// TwinCAT 3 PLC project PLCStudent
// ProgramVersion: 3.1.4022.3
// libraries:
//   Tc2_Standard, * (Beckhoff Automation GmbH)
//   Tc2_System, * (Beckhoff Automation GmbH)
//   Tc3_Module, * (Beckhoff Automation GmbH)
// project tree:
//   GVLs/ GVL.TcGVL
//   / PlcTask.TcTTO
//   POUs/ MAIN.TcPOU, PushPopFB.TcPOU, SFCMotor.TcPOU
// (motion and I/O tree: see PLC project plcsim)
// real-time tasks:
//   TASK PlcTask: cycle T#20ms, priority 20, ADS port 350
// variable links:
//   PLCSim/PLCSim Instance <-> PLCStudent/PLCStudent Instance
//     PlcTask Inputs/GVL.iiDisplayElevat <-> PlcTask Outputs/GVL.qiDispElevat
//     PlcTask Inputs/GVL.ixDoorClose <-> PlcTask Outputs/GVL.qxDoorClose
//     PlcTask Inputs/GVL.ixLampElevat1 <-> PlcTask Outputs/GVL.qxLampElevat1
//     PlcTask Inputs/GVL.ixLampElevat2 <-> PlcTask Outputs/GVL.qxLampElevat2
//     PlcTask Inputs/GVL.ixLampElevat3 <-> PlcTask Outputs/GVL.qxLampElevat3
//     PlcTask Inputs/GVL.ixLampLevel1 <-> PlcTask Outputs/GVL.qxLampLevel1
//     PlcTask Inputs/GVL.ixLampLevel2 <-> PlcTask Outputs/GVL.qxLampLevel2
//     PlcTask Inputs/GVL.ixLampLevel3 <-> PlcTask Outputs/GVL.qxLampLevel3
//     PlcTask Inputs/GVL.ixMotorDown <-> PlcTask Outputs/GVL.qxMotorDown
//     PlcTask Inputs/GVL.ixMotorUp <-> PlcTask Outputs/GVL.qxMotorUp
//     PlcTask Outputs/GVL.qxButtElevat1 <-> PlcTask Inputs/GVL.ixButtElevat1
//     PlcTask Outputs/GVL.qxButtElevat2 <-> PlcTask Inputs/GVL.ixButtElevat2
//     PlcTask Outputs/GVL.qxButtElevat3 <-> PlcTask Inputs/GVL.ixButtElevat3
//     PlcTask Outputs/GVL.qxButtGreen <-> PlcTask Inputs/GVL.ixButtGreen
//     PlcTask Outputs/GVL.qxButtLevel1 <-> PlcTask Inputs/GVL.ixButtLevel1
//     PlcTask Outputs/GVL.qxButtLevel2 <-> PlcTask Inputs/GVL.ixButtLevel2
//     PlcTask Outputs/GVL.qxButtLevel3 <-> PlcTask Inputs/GVL.ixButtLevel3
//     PlcTask Outputs/GVL.qxButtRed <-> PlcTask Inputs/GVL.ixButtRed
//     PlcTask Outputs/GVL.qxDoorClosed <-> PlcTask Inputs/GVL.ixDoorClosed
//     PlcTask Outputs/GVL.qxDoorOpen <-> PlcTask Inputs/GVL.ixDoorOpen
//     PlcTask Outputs/GVL.qxElevatLevel1 <-> PlcTask Inputs/GVL.ixElevatLevel1
//     PlcTask Outputs/GVL.qxElevatLevel2 <-> PlcTask Inputs/GVL.ixElevatLevel2
//     PlcTask Outputs/GVL.qxElevatLevel3 <-> PlcTask Inputs/GVL.ixElevatLevel3

CONFIGURATION PLCStudent
    RESOURCE PLC ON TwinCAT3
        TASK PlcTask(INTERVAL := T#20ms, PRIORITY := 20);
        PROGRAM MAIN WITH PlcTask : MAIN;
    END_RESOURCE
END_CONFIGURATION

// ---- GVLs/GVL.TcGVL
{attribute 'qualified_only'}
VAR_GLOBAL
//Input to PLC from process
	ixButtLevel1		AT %I*:	BOOL;		(* Button at level 1 *)
	ixButtLevel2		AT %I*:	BOOL;		(* Button at level 2 *)
	ixButtLevel3		AT %I*:	BOOL;		(* Button at level 3 *)

	ixButtElevat1		AT %I*:	BOOL;		(* Button 1 inside elevator *)
	ixButtElevat2		AT %I*:	BOOL;		(* Button 2 inside elevator *)
	ixButtElevat3		AT %I*:	BOOL;		(* Button 3 inside elevator *)

	ixButtGreen 		AT %I*:	BOOL;		(* Green button *)
	ixButtRed			AT %I*:	BOOL;		(* Red button, normally closed *)

	ixElevatLevel1 		AT %I*: BOOL;		(* Sensor at level 1 for elevator presence *)
	ixElevatLevel2 		AT %I*: BOOL;		(* Sensor at level 2 for elevator presence *)
	ixElevatLevel3 		AT %I*: BOOL;		(* Sensor at level 3 for elevator presence *)

	ixDoorClosed		AT %I*: BOOL;		(* Sensor for door closed *)
	ixDoorOpen			AT %I*:	BOOL;		(* Sensor for door open *)

//Output from PLC to process
	qxLampLevel1		AT %Q*:	BOOL;		(* Lamp at level 1*)
	qxLampLevel2		AT %Q*:	BOOL;		(* Lamp at level 2*)
	qxLampLevel3		AT %Q*:	BOOL;		(* Lamp at level 3*)

	qxLampElevat1 		AT %Q*:	BOOL;		(* Lamp 1 inside elevator *)
	qxLampElevat2 		AT %Q*:	BOOL;		(* Lamp 2 inside elevator *)
	qxLampElevat3 		AT %Q*:	BOOL;		(* Lamp 3 inside elevator *)

	qxMotorDown			AT %Q*:	BOOL;		(* Run motor down *)
	qxMotorUp			AT %Q*:	BOOL;		(* Run motor up *)

	qxDoorClose			AT %Q*:	BOOL;		(* Close door and keep it closed *)
	qiDispElevat 		AT %Q*:	UINT;		(* Integer display inside elevator *)
END_VAR

// ---- POUs/MAIN.TcPOU
PROGRAM MAIN
VAR
	
END_VAR

SFCMotor();

END_PROGRAM

// ---- POUs/SFCMotor.TcPOU
PROGRAM SFCMotor
VAR
	PushPopFB_0: PushPopFB;
	TargFloor: UINT;
	OutputFloor: UINT;
	MemoryMotor: UINT;

END_VAR
VAR // added by the converter: edge detectors and wires of the graphical bodies
    _rt1, _rt2, _rt3 : R_TRIG;
    _w1, _w2, _w3 : BOOL;
END_VAR

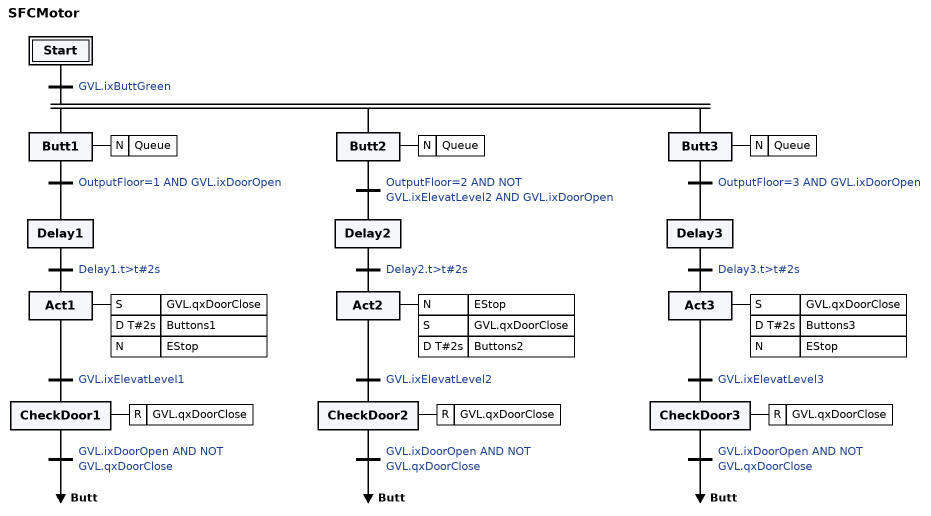
INITIAL_STEP Start:
END_STEP
TRANSITION FROM Start TO (Butt1, Butt2, Butt3)
    := GVL.ixButtGreen;
END_TRANSITION
STEP Butt1:
    Queue(N);
END_STEP
STEP Butt2:
    Queue(N);
END_STEP
TRANSITION FROM Butt2 TO Delay2
    := OutputFloor=2 AND NOT GVL.ixElevatLevel2 AND GVL.ixDoorOpen;
END_TRANSITION
STEP Delay2:
END_STEP
TRANSITION FROM Delay2 TO Act2
    := Delay2.t>t#2s;
END_TRANSITION
STEP Act2:
    EStop(N);
    GVL.qxDoorClose(S);
    Buttons2(D, T#2s);
END_STEP
TRANSITION FROM Act2 TO CheckDoor2
    := GVL.ixElevatLevel2;
END_TRANSITION
STEP CheckDoor2:
    GVL.qxDoorClose(R);
END_STEP
TRANSITION FROM CheckDoor2 TO (Butt1, Butt2, Butt3)
    := GVL.ixDoorOpen AND NOT GVL.qxDoorClose;
END_TRANSITION
STEP Butt3:
    Queue(N);
END_STEP
TRANSITION FROM Butt3 TO Delay3
    := OutputFloor=3 AND GVL.ixDoorOpen;
END_TRANSITION
STEP Delay3:
END_STEP
TRANSITION FROM Delay3 TO Act3
    := Delay3.t>t#2s;
END_TRANSITION
STEP Act3:
    GVL.qxDoorClose(S);
    Buttons3(D, T#2s);
    EStop(N);
END_STEP
TRANSITION FROM Act3 TO CheckDoor3
    := GVL.ixElevatLevel3;
END_TRANSITION
STEP CheckDoor3:
    GVL.qxDoorClose(R);
END_STEP
TRANSITION FROM CheckDoor3 TO (Butt1, Butt2, Butt3)
    := GVL.ixDoorOpen AND NOT GVL.qxDoorClose;
END_TRANSITION
TRANSITION FROM Butt1 TO Delay1
    := OutputFloor=1 AND GVL.ixDoorOpen;
END_TRANSITION
STEP Delay1:
END_STEP
TRANSITION FROM Delay1 TO Act1
    := Delay1.t>t#2s;
END_TRANSITION
STEP Act1:
    GVL.qxDoorClose(S);
    Buttons1(D, T#2s);
    EStop(N);
END_STEP
TRANSITION FROM Act1 TO CheckDoor1
    := GVL.ixElevatLevel1;
END_TRANSITION
STEP CheckDoor1:
    GVL.qxDoorClose(R);
END_STEP
TRANSITION FROM CheckDoor1 TO (Butt1, Butt2, Butt3)
    := GVL.ixDoorOpen AND NOT GVL.qxDoorClose;
END_TRANSITION
// branch label Butt

ACTION Buttons1:

IF GVL.ixDoorClosed THEN
	
	IF GVL.ixElevatLevel2 OR GVL.ixElevatLevel3 THEN
		GVL.qxMotorDown := TRUE;
	END_IF

	IF GVL.ixElevatLevel1  THEN
		GVL.qxMotorDown :=FALSE;
		GVL.qxMotorUp :=FALSE;
	END_IF
END_IF
END_ACTION

ACTION Buttons2:
IF GVL.ixDoorClosed THEN
	IF GVL.ixElevatLevel1 THEN
		GVL.qxMotorUp := TRUE;
	END_IF

	IF GVL.ixElevatLevel3  THEN
		GVL.qxMotorDown :=TRUE;
	END_IF

	IF GVL.ixElevatLevel2  THEN
		GVL.qxMotorDown :=FALSE;
		GVL.qxMotorUp :=FALSE;
	END_IF
END_IF
END_ACTION

ACTION Buttons3:
IF GVL.ixDoorClosed THEN
	
	IF GVL.ixElevatLevel2 OR GVL.ixElevatLevel1 THEN
		GVL.qxMotorUp := TRUE;
	END_IF

	IF GVL.ixElevatLevel3  THEN
		GVL.qxMotorDown :=FALSE;
		GVL.qxMotorUp :=FALSE;
	END_IF
END_IF
END_ACTION

ACTION CheckDoor:


IF GVL.ixDoorClosed THEN
	GVL.qxDoorClose := FALSE;
END_IF
END_ACTION

ACTION EStop:


IF NOT GVL.ixButtRed  THEN
	IF GVL.qxMotorDown THEN
		GVL.qxMotorDown :=FALSE;
		MemoryMotor :=2;
	
	ELSIF GVL.qxMotorUp THEN
		GVL.qxMotorUp :=FALSE;
		MemoryMotor :=1;
	
	END_IF
END_IF

IF GVL.ixButtGreen AND MemoryMotor>0 THEN
	IF OutputFloor=2 AND MemoryMotor=1 THEN
		GVL.qxMotorUp:=TRUE;
		MemoryMotor:=0;
	END_IF

	IF OutputFloor=2 AND MemoryMotor=2 THEN
		GVL.qxMotorDown:=TRUE;
		MemoryMotor:=0;
	END_IF

	IF OutputFloor=1 AND MemoryMotor=2 THEN
		GVL.qxMotorDown:=TRUE;
		MemoryMotor:=0;
	END_IF

	IF OutputFloor=3 AND MemoryMotor=1 THEN
		GVL.qxMotorUp:=TRUE;
		MemoryMotor:=0;
	END_IF
END_IF
END_ACTION

ACTION Queue:
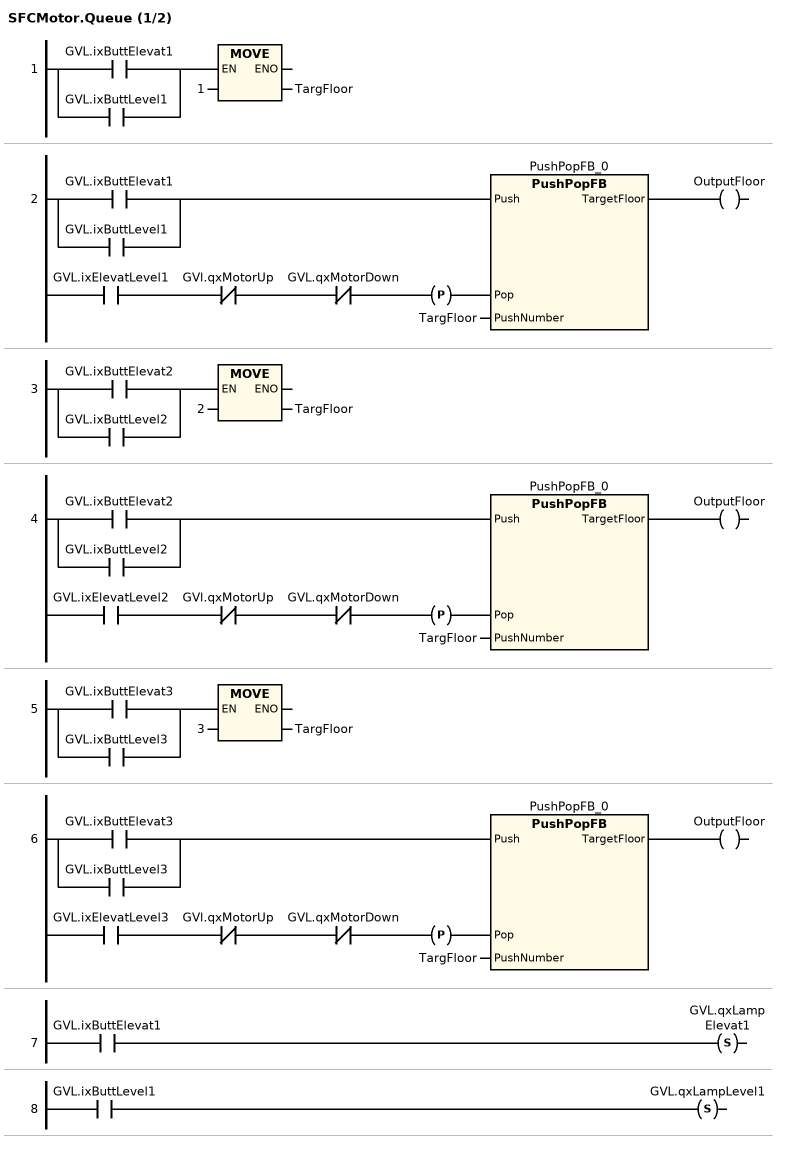
// NETWORK 1
IF GVL.ixButtElevat1 OR GVL.ixButtLevel1 THEN TargFloor := 1; END_IF

// NETWORK 2
_rt1(CLK := GVL.ixElevatLevel1 AND NOT GVl.qxMotorUp AND NOT GVL.qxMotorDown);
PushPopFB_0(Push := GVL.ixButtElevat1 OR GVL.ixButtLevel1, Pop := _rt1.Q, PushNumber := TargFloor); // PushPopFB
OutputFloor := PushPopFB_0.TargetFloor;

// NETWORK 3
IF GVL.ixButtElevat2 OR GVL.ixButtLevel2 THEN TargFloor := 2; END_IF

// NETWORK 4
_rt2(CLK := GVL.ixElevatLevel2 AND NOT GVl.qxMotorUp AND NOT GVL.qxMotorDown);
PushPopFB_0(Push := GVL.ixButtElevat2 OR GVL.ixButtLevel2, Pop := _rt2.Q, PushNumber := TargFloor); // PushPopFB
OutputFloor := PushPopFB_0.TargetFloor;

// NETWORK 5
IF GVL.ixButtElevat3 OR GVL.ixButtLevel3 THEN TargFloor := 3; END_IF

// NETWORK 6
_rt3(CLK := GVL.ixElevatLevel3 AND NOT GVl.qxMotorUp AND NOT GVL.qxMotorDown);
PushPopFB_0(Push := GVL.ixButtElevat3 OR GVL.ixButtLevel3, Pop := _rt3.Q, PushNumber := TargFloor); // PushPopFB
OutputFloor := PushPopFB_0.TargetFloor;

// NETWORK 7
GVL.qxLampElevat1 S= GVL.ixButtElevat1;

// NETWORK 8
GVL.qxLampLevel1 S= GVL.ixButtLevel1;

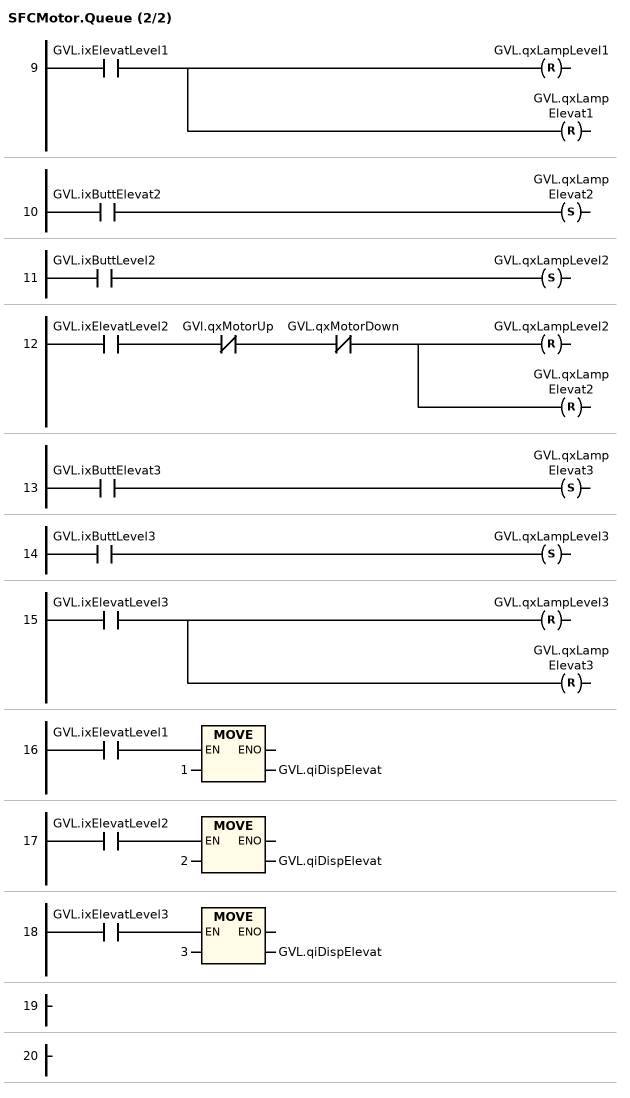
// NETWORK 9
_w1 := GVL.ixElevatLevel1;
GVL.qxLampLevel1 R= _w1;
GVL.qxLampElevat1 R= _w1;

// NETWORK 10
GVL.qxLampElevat2 S= GVL.ixButtElevat2;

// NETWORK 11
GVL.qxLampLevel2 S= GVL.ixButtLevel2;

// NETWORK 12
_w2 := GVL.ixElevatLevel2 AND NOT GVl.qxMotorUp AND NOT GVL.qxMotorDown;
GVL.qxLampLevel2 R= _w2;
GVL.qxLampElevat2 R= _w2;

// NETWORK 13
GVL.qxLampElevat3 S= GVL.ixButtElevat3;

// NETWORK 14
GVL.qxLampLevel3 S= GVL.ixButtLevel3;

// NETWORK 15
_w3 := GVL.ixElevatLevel3;
GVL.qxLampLevel3 R= _w3;
GVL.qxLampElevat3 R= _w3;

// NETWORK 16
IF GVL.ixElevatLevel1 THEN GVL.qiDispElevat := 1; END_IF

// NETWORK 17
IF GVL.ixElevatLevel2 THEN GVL.qiDispElevat := 2; END_IF

// NETWORK 18
IF GVL.ixElevatLevel3 THEN GVL.qiDispElevat := 3; END_IF

// NETWORK 19

// NETWORK 20
END_ACTION

END_PROGRAM

// ---- POUs/PushPopFB.TcPOU
FUNCTION_BLOCK PushPopFB
VAR_INPUT
	Push:BOOL;
	Pop: BOOL;
	PushNumber: UINT;
END_VAR
VAR_OUTPUT
	TargetFloor: UINT;
END_VAR
VAR
	Queue: ARRAY [1..3] OF UINT:=[0,0,0];
	numberExist : BOOL;
	i: INT:=1;
END_VAR



IF Push THEN
    numberExist := FALSE;
    FOR i:=1 TO 3 DO
        IF Queue[i] = PushNumber THEN
            numberExist := TRUE;
            EXIT; // Exit as soon as a duplicate is found
        END_IF
    END_FOR

    IF NOT numberExist THEN
        FOR i:=1 TO 3 DO
            IF Queue[i] = 0 THEN
                Queue[i] := PushNumber;
                EXIT; // Exit after inserting the number to the first empty slot
            END_IF
        END_FOR
    END_IF
END_IF



IF Pop THEN
	FOR i:=1 TO 2 DO
		Queue[i]:=Queue[i+1];
	END_FOR
	Queue[3]:=0;
END_IF


// Store Target Floor

FOR i:=1 TO 3 DO
	IF Queue[i] <> 0 THEN
		TargetFloor := Queue[i];
		EXIT;
	END_IF
END_FOR

END_FUNCTION_BLOCK
